FUNCTION_BLOCK OpcUaCreateId (* Creates an OPC UA identifier *)
  (* Standard: 61499-2; Description: Copyright (c) 2026 Monika Wenger This program and the accompanying materials are made available under the terms of the Eclipse Public License 2.0 which is available at https://www.eclipse.org/legal/epl-2.0/ SPDX-License-Identifier: EPL-2.0 *)
  (* Version 3.0, 2025-12-05, Monika Wenger *)
  PACKAGE eclipse4diac::opcua;
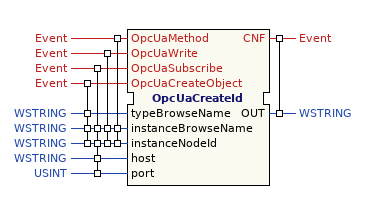
  EVENT_INPUT
    OpcUaMethod WITH instanceBrowseName, instanceNodeId;
    OpcUaWrite WITH instanceBrowseName, instanceNodeId;
    OpcUaSubscribe WITH instanceBrowseName, instanceNodeId, host, port;
    OpcUaCreateObject WITH typeBrowseName, instanceBrowseName, instanceNodeId;
  END_EVENT
  EVENT_OUTPUT
    CNF WITH OUT;
  END_EVENT
  VAR_INPUT
    typeBrowseName : WSTRING;
    instanceBrowseName : WSTRING;
    instanceNodeId : WSTRING;
    host : WSTRING;
    port : USINT;
  END_VAR
  VAR_OUTPUT
    OUT : WSTRING;
  END_VAR
  VAR CONSTANT
    PREFIX : WSTRING := "opc_ua[";
    SUFFIX : WSTRING := "]";
    OPCUA_CREATE_METHOD : WSTRING := "CREATE_METHOD;";
    OPCUA_WRITE : WSTRING := "WRITE;";
    OPCUA_SUBSCRIBE : WSTRING := "SUBSCRIBE;opc.tcp://";
    OPCUA_CREATE_OBJECT : WSTRING := "CREATE_OBJECT;";
    NODEID_TYPE : WSTRING := ",s=";
    SEPARATOR_PAIR : WSTRING := ";";
    SEPARATOR_HOST : WSTRING := ":";
    SEPARATOR_HASH : WSTRING := "#;";
  END_VAR
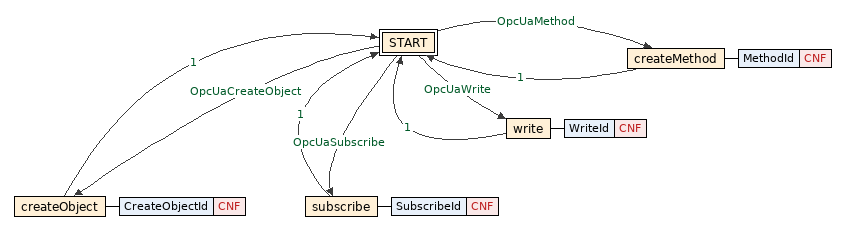
  EC_STATES
    START; (* Initial State *)
    createMethod : MethodId -> CNF;
    write : WriteId -> CNF;
    subscribe : SubscribeId -> CNF;
    createObject : CreateObjectId -> CNF;
  END_STATES
  EC_TRANSITIONS
    START TO createMethod := OpcUaMethod;
    createMethod TO START := 1;
    START TO write := OpcUaWrite;
    write TO START := 1;
    START TO subscribe := OpcUaSubscribe;
    subscribe TO START := 1;
    START TO createObject := OpcUaCreateObject;
    createObject TO START := 1;
  END_TRANSITIONS
  ALGORITHM MethodId IN ST:
OUT := CONCAT(PREFIX, OPCUA_CREATE_METHOD, instanceBrowseName, NODEID_TYPE, instanceNodeId, SUFFIX);
  END_ALGORITHM
  ALGORITHM WriteId IN ST:
OUT := CONCAT(PREFIX, OPCUA_WRITE, instanceBrowseName, NODEID_TYPE, instanceNodeId, SUFFIX);
  END_ALGORITHM
  ALGORITHM SubscribeId IN ST:
OUT := CONCAT(PREFIX, OPCUA_SUBSCRIBE, host, SEPARATOR_HOST, USINT_AS_WSTRING(port), SEPARATOR_HASH, instanceBrowseName,
	NODEID_TYPE, instanceNodeId, SUFFIX);
  END_ALGORITHM
  ALGORITHM CreateObjectId IN ST:
OUT := CONCAT(PREFIX, OPCUA_CREATE_OBJECT, typeBrowseName, SEPARATOR_PAIR, instanceBrowseName, NODEID_TYPE,
	instanceNodeId, SUFFIX);
  END_ALGORITHM
END_FUNCTION_BLOCK
